(* IEC 61131-3 sources: sps_maggio25/src, 4 files *)

(* ---- LGF_Random_Real.st ---- *)
USING Siemens.Simatic.S71500.Clocks;
USING System.DateTime;
NAMESPACE ProgramEdge

    TYPE
        DTL : STRUCT
            YEAR : UINT;
            MONTH : USINT;
            DAY : USINT;
            WEEKDAY : USINT;
            HOUR : USINT;
            MINUTE : USINT;
            SECOND : USINT;
            NANOSECOND : UDINT;
        END_STRUCT;
    END_TYPE

    FUNCTION LGF_Random_Real : REAL
        VAR_EXTERNAL CONSTANT
            ZERO : REAL;
            MAX_UDINT : UDINT;
            SUB_STATUS_NO_ERROR : WORD;
            STATUS_FINISHED_NO_ERROR : WORD;
            ERR_RD_SYS_T : WORD;
        END_VAR

        VAR_OUTPUT
            error : BOOL;
            status : WORD;
            subfunctionStatus : WORD;
        END_VAR

        VAR_TEMP
            //tempTime : DTL;
            tempTime : LDATE_AND_TIME;
            tempTimeNanoSecond : INT;
            tempNanoSecondInDWord : DWORD;
            tempTimeStatus : WORD;
            tempRandomValue : DWORD;
        END_VAR
        ;

    // Read system time
    GetSystemDateTime(value => tempTime);

    //non abbiamo ritorno
    // Check return variable for error
    /*IF (tempTimeStatus <> SUB_STATUS_NO_ERROR) THEN
        error := true;
        status := ERR_RD_SYS_T;
        subfunctionStatus := tempTimeStatus;
        LGF_Random_Real := ZERO;
        RETURN;
    END_IF;*/

    SplitDateAndTime(
            value := tempTime,
            nanosecond => tempTimeNanoSecond
        );

    // Converting to double word so individual bytes can be addressed
    tempNanoSecondInDWord := TO_DWORD(tempTimeNanoSecond);

    // Calculate a random-start-value depending on the time
    tempRandomValue.%B3 := tempNanoSecondInDWord.%B0;
    tempRandomValue.%B2 := tempNanoSecondInDWord.%B1;
    tempRandomValue.%B1 := tempNanoSecondInDWord.%B2;
    tempRandomValue.%B0 := tempNanoSecondInDWord.%B3;

    // Norm the calculated random number: 0.0 <= Random_Real <= 1.0
    LGF_Random_Real := TO_REAL(TO_UDINT(tempRandomValue)) / TO_REAL(MAX_UDINT);

    error := false;
    status := STATUS_FINISHED_NO_ERROR;
    subfunctionStatus := SUB_STATUS_NO_ERROR;

    END_FUNCTION
END_NAMESPACE

(* ---- GetTimeStamp.st ---- *)
USING Siemens.Simatic.S71500.Clocks;
NAMESPACE ProgramEdge
    FUNCTION GetTimeStamp : INT
        // Function GetTimestamp

        VAR_TEMP
            actDT : LDATE_AND_TIME; // in TIA era Date_and_Time
            TS : LINT; //in TIA era ULINT
            diffLTime : LTime;
            retVal : Int;
            retValRD_LOC_T : Int;
        END_VAR

        VAR_OUTPUT
            Timestamp : UDInt;
        END_VAR

        TS := LINT#0;

        //in TIA
        //retValRD_LOC_T := RD_LOC_T(OUT => TIAactDT);

        retValRD_LOC_T := TO_INT(GetLocalDateTime(value => actDT));

        IF  retValRD_LOC_T = 0 OR retValRD_LOC_T = 1 THEN

            //in TIA
            //diffLTime := T_DIFF_LTIME(IN1 := TO_LDT(actDT), IN2 := LDT#2020-01-01-00:00:00.0);
            diffLTime := actDT - LDT#2020-01-01-00:00:00.0;
            TS := TO_LINT(diffLTime) / LINT#1000000000;
            retVal := 0;
        ELSE
            retVal := 1;
        END_IF;

        Timestamp := TO_UDINT(TS);
        GetTimestamp := retVal;

    END_FUNCTION
END_NAMESPACE

(* ---- configuration.st ---- *)
USING Siemens.Simatic.S71500.Tasks;
USING ProgramModuli;

//{OpcUa.NodeGenerator.IdType = SymbolName}
CONFIGURATION MyConfiguration
    TASK Main (Priority := 1);
    TASK MyInterruptTask : CyclicInterrupt := (
        CycleTime := T#500ms,
        EventPriority := USINT#13
    );

    PROGRAM P1 WITH Main : MainProgram;
    PROGRAM P2 WITH MyInterruptTask : ProgramCycling;

    {S7.extern = ReadWrite}
//    {OpcUa.AccessLevel = ReadWrite}
    VAR_GLOBAL
        GoodPieces : DINT;
        BadPieces : DINT;
        MachSpeed : REAL;
        MachSpeedSeconds : REAL;
        RejectRatio : REAL;
        MachineStatus : INT := 1;
        TotalPieces : DINT;
        SetpointSpeedSeconds : REAL;
        SetpointSpeed : REAL;
        TimeT : REAL;
        TimeStarted : REAL;
        TimeStopped : REAL;
        LastTimeStopped : REAL;
        LastTimeStarted : REAL;
        LastTimeMaintenance : REAL;
        ProductionActive : BOOL;
        TotalActiveEnergy : LREAL;
        OilLevel : REAL := REAL#100.0;
        ResetOilLevel : BOOL;
        BatchNum : UDINT;
        BatchPieces : DINT := 7000;
        BatchProductName : String := 'Product_C';
        ProductNames : Array[0..3] of String := ['Product_A', 'Product_B', 'Product_C', 'Product_D'];
        BatchBadPieces : DINT;
        BatchGoodPieces : DINT;
        BatchTotalPieces : DINT;
    END_VAR

    VAR_GLOBAL CONSTANT
        EnergyConsumptionStarted : REAL := REAL#0.0417;
        EnergyConsumptionHold : REAL := REAL#0.0152;
        EnergyConsumptionMaintenance : REAL := REAL#0.0121;
        EnergyConsumptionStopped : REAL := REAL#0.0243;
        MaxReal : REAL := REAL#1.234567e+20;
        MaxDInt : DINT := DINT#2147483647;
    END_VAR

    VAR_GLOBAL CONSTANT
        ZERO : REAL := REAL#0.0;
        MAX_UDINT : UDINT := UDINT#4294967295;
        SUB_STATUS_NO_ERROR : WORD := WORD#16#0000;
        STATUS_FINISHED_NO_ERROR : WORD := WORD#16#0000;
        ERR_RD_SYS_T : WORD := WORD#16#8600;
    END_VAR

    VAR_GLOBAL
        {S7.extern = ReadWrite}
        {OpcUa.AccessLevel=ReadWrite}
        enable: BOOL;

        tank : Tank;

        ctrlInletOpen AT %Q0.0: BOOL;
        ctrlOutletOpen AT %Q0.1: BOOL;
    END_VAR

END_CONFIGURATION

(* ---- program.st ---- *)
USING System.Conversion;
USING ProgramEdge;

PROGRAM ProgramCycling

    VAR_EXTERNAL CONSTANT
        EnergyConsumptionStarted : REAL;
        EnergyConsumptionHold : REAL;
        EnergyConsumptionMaintenance : REAL;
        EnergyConsumptionStopped : REAL;
        MaxReal : REAL;
        MaxDInt : DINT;
    END_VAR

    VAR_EXTERNAL
        GoodPieces : DINT;
        BadPieces : DINT;
        MachSpeed : REAL;
        MachSpeedSeconds : REAL;
        RejectRatio : REAL;
        MachineStatus : INT;
        TotalPieces : DINT;
        SetpointSpeedSeconds : REAL;
        SetpointSpeed : REAL;
        TimeT : REAL;
        TimeStarted : REAL;
        TimeStopped : REAL;
        LastTimeStopped : REAL;
        LastTimeStarted : REAL;
        LastTimeMaintenance : REAL;
        ProductionActive : BOOL;
        TotalActiveEnergy : LREAL;
        OilLevel : REAL;
        ResetOilLevel : BOOL;
        BatchNum : UDINT;
        BatchPieces : DINT;
        BatchProductName : STRING;
        ProductNames : ARRAY [0..3] OF STRING;
        BatchBadPieces : DINT;
        BatchGoodPieces : DINT;
        BatchTotalPieces : DINT;
    END_VAR

    VAR_TEMP
        MachSpeedInACycle : REAL;
        RandomErr : BOOL;
        RandomStatus : WORD;
        RandomSubStatus : WORD;
        InternalVal : REAL;
        RandomVal : REAL;
        RandomTime : REAL;
        RandomSign : INT;
        RandomProductIndex : INT;
        retVal : INT;
    END_VAR

// get random value from 0.0 to 1.0
RandomVal := LGF_Random_Real(error => RandomErr, status => RandomStatus, subfunctionStatus => RandomSubStatus);
// get random sign based on randomval
IF RandomVal >= 0.6 THEN
    RandomSign := -1;
ELSE
    RandomSign := 1;
END_IF;
// if total batch pieces are reach close the batch
// and start new batch
IF BatchTotalPieces >= BatchPieces
    OR BatchNum = UDINT#0 THEN
    // reset pieces
    BatchBadPieces := 0;
    BatchGoodPieces := 0;
    BatchTotalPieces := 0;
    // set batch num as actual epoch
    retVal := GetTimestamp(BatchNum);
    // get random value from 0.0 to 1.0
    RandomVal := LGF_Random_Real(error => RandomErr, status => RandomStatus, subfunctionStatus => RandomSubStatus);
    // get a random number of pieces for new batch
    BatchPieces := 10000 + TO_INT(3000 * RandomVal * RandomSign);
    // based on random val get a product index
    // and set to batch product name
    InternalVal:= (TO_INT (RandomVal * 100) / 4);
    RandomProductIndex := TO_INT(RandomVal * 100)- (4 * TO_INT(InternalVal));
    BatchProductName := ProductNames[RandomProductIndex];
    // put machine in stopped status
    MachineStatus := 0;
END_IF;

//
// increment production time
TimeT := TimeT + REAL#0.5;
IF MachineStatus = 1 THEN
    TimeStarted := TimeStarted + REAL#0.5;
ELSE
    TimeStopped := TimeStopped + REAL#0.5;
END_IF;
// reset time when max reached
IF TimeT >= MaxReal THEN
    TimeT := REAL#0.0;
    TimeStarted := REAL#0.0;
    TimeStopped := REAL#0.0;
END_IF;

//
// get random value from 0.0 to 1.0
RandomVal := LGF_Random_Real(error => RandomErr, status => RandomStatus, subfunctionStatus => RandomSubStatus);
// get random sign based on randomval
IF RandomVal >= 0.6 THEN
    RandomSign := -1;
ELSE
    RandomSign := 1;
END_IF;

// get a random time 2000 +- 300sec
RandomTime := 2000 + (RandomVal * 300 *RandomSign);
// if the time since machine is started is enough
// try to change machine mode to hold or stopped
IF TimeT - LastTimeStarted > RandomTime THEN
    IF RandomVal >= 0.64 AND RandomVal < 0.74 THEN
        IF MachineStatus = 1 THEN
            // started -> hold
            MachineStatus := 2;
            LastTimeStarted := TimeT;
        END_IF;
    ELSIF RandomVal >= 0.3 AND RandomVal < 0.4 THEN
        IF MachineStatus = 1 THEN
            // started -> stopped
            MachineStatus := 0;
            LastTimeStarted := TimeT;
        END_IF;
    END_IF;
END_IF;

// get a random time 5000 +- 1000sec
RandomTime := 5000 + (RandomVal * 1000 * RandomSign);
// if the time since machine is started is enough,
// try to change machine mode to maintenance
IF TimeT - LastTimeMaintenance > RandomTime THEN
    IF RandomVal >= 0.61 AND RandomVal < 0.84 THEN
        IF MachineStatus = 1 THEN
            // started -> maintenance
            MachineStatus := 3;
            LastTimeMaintenance := TimeT;
        END_IF;
    END_IF;
END_IF;

// get a random time 1000 +- 200sec
RandomTime := 1000 + (RandomVal * 200 * RandomSign);
// if the time since machine is stopped is enough, try to change machine mode
IF TimeT - LastTimeStopped > RandomTime THEN
    IF RandomVal >= 0.25 AND RandomVal < 0.32 THEN
        IF MachineStatus = 2 THEN
            // hold -> started
            MachineStatus := 1;
            LastTimeStopped := TimeT;
        END_IF;
    ELSIF RandomVal >= 0.45 AND RandomVal < 0.52 THEN
        IF MachineStatus = 3 THEN
            // maintenance -> started
            MachineStatus := 1;
            LastTimeStopped := TimeT;
        END_IF;
    ELSIF RandomVal >= 0.71 AND RandomVal < 0.81 THEN
        IF MachineStatus = 0 THEN
            // stopped -> started
            MachineStatus := 1;
            LastTimeStopped := TimeT;
        END_IF;
    END_IF;
END_IF;

//
// change setpoint speed
IF SetpointSpeed <= 360.0 AND RandomVal >= 0.1 AND RandomVal < 0.15 THEN
    // increase or decrease setpoint
    SetpointSpeed := (SetpointSpeed + REAL#10.0)*RandomSign;
ELSIF SetpointSpeed > 360.0 THEN
    // reset setpoint
    SetpointSpeed := REAL#359.0;
ELSIF SetpointSpeed < 120.0 THEN
    // min limit of machine speed
    SetpointSpeed := REAL#120.0;
END_IF;

//
// based on machine status
IF MachineStatus = 1 THEN
    // if machine is started
    IF MachSpeed < 120 THEN
        // min limit of machine speed
        MachSpeed := 120;
    END_IF;
    // check production speed
    IF MachSpeed <= SetpointSpeed THEN
        // min limit of machine speed
        MachSpeed := MachSpeed +
        (SetpointSpeed - MachSpeed) * REAL#0.75;
    ELSIF MachSpeed > SetpointSpeed THEN
        // max limit of machine speed
        MachSpeed := SetpointSpeed;
    END_IF;
    // change reject ratio
    IF RejectRatio <= 0.25 THEN
        // increase
        RejectRatio := RejectRatio + REAL#0.05;
    ELSIF RejectRatio > 0.25 THEN
        // reset to min
        RejectRatio := REAL#0.0;
    END_IF;
    // get production ratio in a cycle from pcs/min (every 500 ms)
    MachSpeedInACycle := MachSpeed / REAL#120.0;
    // update speeds in sec
    SetpointSpeedSeconds := SetpointSpeed / REAL#60.0;
    MachSpeedSeconds := MachSpeed / REAL#60.0;
    // status boolean for started status
    ProductionActive := TRUE;

    // get random value from 0.0 to 1.0
    RandomVal := LGF_Random_Real(error => RandomErr, status => RandomStatus, subfunctionStatus => RandomSubStatus);
    IF RandomVal < RejectRatio THEN
        // if random < probability of bad production make bad pieces
        BadPieces := BadPieces + TO_DINT(Ceil(MachSpeedInACycle));
        BatchBadPieces := BatchBadPieces + TO_DINT(Ceil(MachSpeedInACycle));
    ELSE
        // else make good pieces
        GoodPieces := GoodPieces + TO_DINT(Ceil(MachSpeedInACycle));
        BatchGoodPieces := BatchGoodPieces + TO_DINT(Ceil(MachSpeedInACycle));
    END_IF;
    // update total
    TotalPieces := GoodPieces + BadPieces;
    BatchTotalPieces := BatchGoodPieces + BatchBadPieces;

    // reset pieces when reach max
    IF TotalPieces > MaxDInt THEN
        BatchBadPieces := 0;
        BatchGoodPieces := 0;
       END_IF;

ELSIF MachineStatus = 3 THEN
    // update machspeedsec
    SetpointSpeedSeconds := REAL#0.0;
    SetpointSpeed := REAL#0.0;
    // reset speed
    MachSpeed := REAL#0.0;
    MachSpeedSeconds := REAL#0.0;
    // status boolean for started status
    ProductionActive := FALSE;
ELSE
    // reset speed
    MachSpeed := REAL#0.0;
    MachSpeedSeconds := REAL#0.0;
    // status boolean for started status
    ProductionActive := FALSE;
END_IF;

//
// Energy Consumption based on status
IF MachineStatus = 0 THEN
    TotalActiveEnergy := TotalActiveEnergy + EnergyConsumptionStopped;
ELSIF MachineStatus = 1 THEN
    TotalActiveEnergy := TotalActiveEnergy + EnergyConsumptionStarted;
ELSIF MachineStatus = 2 THEN
    TotalActiveEnergy := TotalActiveEnergy + EnergyConsumptionHold;
ELSIF MachineStatus = 3 THEN
    TotalActiveEnergy := TotalActiveEnergy + EnergyConsumptionMaintenance;
END_IF;
// reset energy on max
IF TotalActiveEnergy >= MaxReal THEN
    TotalActiveEnergy := 0;
END_IF;

//
// get random value from 0.0 to 1.0
RandomVal := LGF_Random_Real(error => RandomErr, status => RandomStatus, subfunctionStatus => RandomSubStatus);
// OIL Level consumption in production
IF MachineStatus = 1 THEN
    IF RandomVal >= 0.9 AND RandomVal <= 1.0 THEN
        OilLevel := OilLevel - REAL#0.00001;
    ELSIF RandomVal >= 0.4 AND RandomVal < 0.7 THEN
        OilLevel := OilLevel - REAL#0.000006;
    ELSIF RandomVal >= 0.1 AND RandomVal < 0.4 THEN
        OilLevel := OilLevel - REAL#0.000002;
    END_IF;
END_IF;
// OIL Level Reset trigger
IF ResetOilLevel = TRUE THEN
    OilLevel := REAL#100.0;
    ResetOilLevel := FALSE;
END_IF;

END_PROGRAM
